FUNCTION_BLOCK GAUSSIANBLUR (* openCV gaussian blur filter *)
  (* Version 1.0, AN, SWDC RTSoft *)
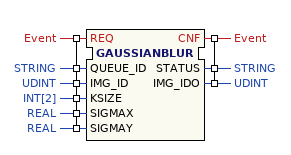
  EVENT_INPUT
    REQ WITH QUEUE_ID, IMG_ID, KSIZE, SIGMAX, SIGMAY;
  END_EVENT
  EVENT_OUTPUT
    CNF WITH STATUS, IMG_IDO;
  END_EVENT
  VAR_INPUT
    QUEUE_ID : STRING;
    IMG_ID : UDINT;
    KSIZE : ARRAY [0..1] OF INT; (* Gaussian kernel size (width, height) *)
    SIGMAX : REAL; (* kernel deviation in X direction *)
    SIGMAY : REAL; (* kernel deviation in Y direction *)
  END_VAR
  VAR_OUTPUT
    STATUS : STRING;
    IMG_IDO : UDINT;
  END_VAR
  ALGORITHM REQ IN ST:

  END_ALGORITHM
END_FUNCTION_BLOCK
